(* PLC project Unnamed, Unknown Unnamed 1 *)
(* stored: creationDateTime 2025-10-31T14:35:28, modificationDateTime 2025-10-31T15:04:53 *)

PROGRAM program0
  VAR
    Sensor : BOOL;
    Flag : BOOL;
    Count : INT := 1;
    One : INT := 1;
    Two : INT := 2;
    TON0 : TON;
  END_VAR
  VAR  (* added by the conversion: wires and edge detectors of the diagram *)
    _GE6_OUT : BOOL;
  END_VAR

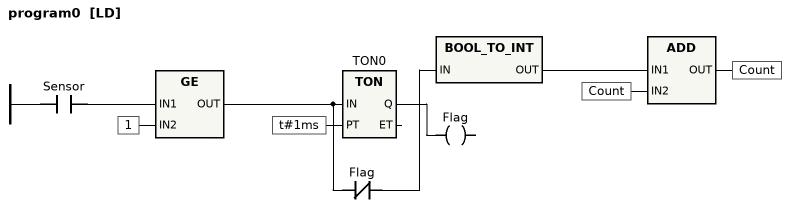
(* LD diagram, written out as Structured Text *)
_GE6_OUT := Sensor >= 1;
Count := BOOL_TO_INT(_GE6_OUT AND NOT Flag) + Count;
TON0(IN := _GE6_OUT, PT := t#1ms);
Flag := TON0.Q;
END_PROGRAM

CONFIGURATION Config0
  RESOURCE Res0 ON PLC
    TASK task0(INTERVAL := T#20ms, PRIORITY := 0);
    PROGRAM instance0 WITH task0 : program0;
  END_RESOURCE
END_CONFIGURATION
